PROGRAM MAIN
VAR
END_VAR

END_PROGRAM

(* stored: Version 1.1.0.1
   POU MAIN: Id {0f0b6438-34c2-45c8-a3bc-603e78d55c99} *)
